INTERFACE I_ParamMediator

(*
  Release deformation ct
  TODO: find another way to do inter worker communication for generic methods.
*)
METHOD ClearCachedCT
VAR_INPUT
  iCT              : I_CT;
END_VAR
END_METHOD

{attribute 'monitoring':='call'}
PROPERTY fCameraToPrintOffset : LREAL
GET
END_GET
END_PROPERTY

{attribute 'monitoring':='call'}
PROPERTY fDetectToCamera : LREAL
GET
END_GET
END_PROPERTY

(*
  Distance (Offset) from Master-Trigger to Master Reference Position.
  NOTE: This is normally the distance between the first (MASTER) StartPosDetection to first print Module (Printing Unit) 
*)
PROPERTY fMasterDetectToRefPos : LREAL
GET
END_GET
END_PROPERTY

METHOD init
VAR_INPUT
  pCreateWorker : POINTER TO FB_WorkerDefGrid_Python;
  pCamWorker : POINTER TO FB_WorkerDefGrid_Camera;
  pDefWorker : POINTER TO FB_WorkerDefGrid_Deformation;
END_VAR
END_METHOD

PROPERTY sCameraGridSettings : ST_CameraGridSettings
GET
END_GET
END_PROPERTY

PROPERTY sDeformationGridSetttings : ST_DefGridSettings
GET
END_GET
END_PROPERTY

END_INTERFACE

(* stored: Version 1.1.0.1, ProductVersion 3.1.4024.11
   Itf I_ParamMediator: Id {44f2ddfb-07a7-4305-bf98-9eca0b2e7285}
   Method ClearCachedCT: Id {37ede8fa-36b6-4e30-8b33-b7c3259ebe07}
   Property fCameraToPrintOffset: Id {89859152-e725-4920-abf7-677c2007ee9c}
   Get Get: Id {2fc6b5ef-b27a-4835-a6b5-a72f5d7d8629}
   Property fDetectToCamera: Id {11ad5319-cf27-4b8b-81be-9a27f3c64a75}
   Get Get: Id {478f1e90-b6a4-4e92-9b77-809f2c0ab59d}
   Property fMasterDetectToRefPos: Id {c872806f-01d3-44f9-baa0-4643b95ecb2c}
   Get Get: Id {2ffe41b5-235e-45e6-a44a-44363033cc23}
   Method init: Id {9b7c392c-bc43-4afa-b5f3-a650552ff470}
   Property sCameraGridSettings: Id {f28e61e7-9fce-4611-bc89-520b4efc0649}
   Get Get: Id {fa4b007d-6456-4d0f-9d70-1d8af69098e5}
   Property sDeformationGridSetttings: Id {ecefed7e-560d-422a-a3ff-1a9e4e97de76}
   Get Get: Id {4bb826c1-2467-45c1-99fb-cdadf553de78} *)
